INTERFACE I_Pump EXTENDS I_ComponentBase

PROPERTY Speed : LREAL
GET
END_GET
SET
END_SET
END_PROPERTY

METHOD Start : BOOL
VAR_INPUT
END_VAR
END_METHOD

METHOD Stop
VAR_INPUT
END_VAR
END_METHOD

END_INTERFACE

(* stored: Version 1.1.0.1
   Itf I_Pump: Id {d78329b0-a379-4c56-b3ca-f9a2852ddf70}
   Property Speed: Id {e17b8117-c438-4504-8a36-37d094e1b151}
   Get Get: Id {b0fb3859-fd3e-43c7-bf9d-6c5e78830cbc}
   Set Set: Id {a519748c-697d-4b21-b608-ed0fdacc2b50}
   Method Start: Id {b65a9d77-77cd-4864-b72f-c075c548bcb5}
   Method Stop: Id {f6f9a771-cf2b-44bb-8862-463f7d17dd3f} *)
